// TIA Portal V19 export
FUNCTION_BLOCK "Dispenser_Main"   // FB1, LAD
TITLE = Main Block for Dispenser Element and Conveyor Running
{ S7_Optimized_Access := 'TRUE' }
// Holds Code for Dispenser Project , Light Gates and Conveyor Belt Motor.
// stored: MemoryReserve 100, SetENOAutomatically false
   VAR_TEMP   // added for the SCL form of the ladder/FBD networks
      _w1 : Bool;
   END_VAR
BEGIN

REGION Network 1: Power Up
   // Enabled Power To System
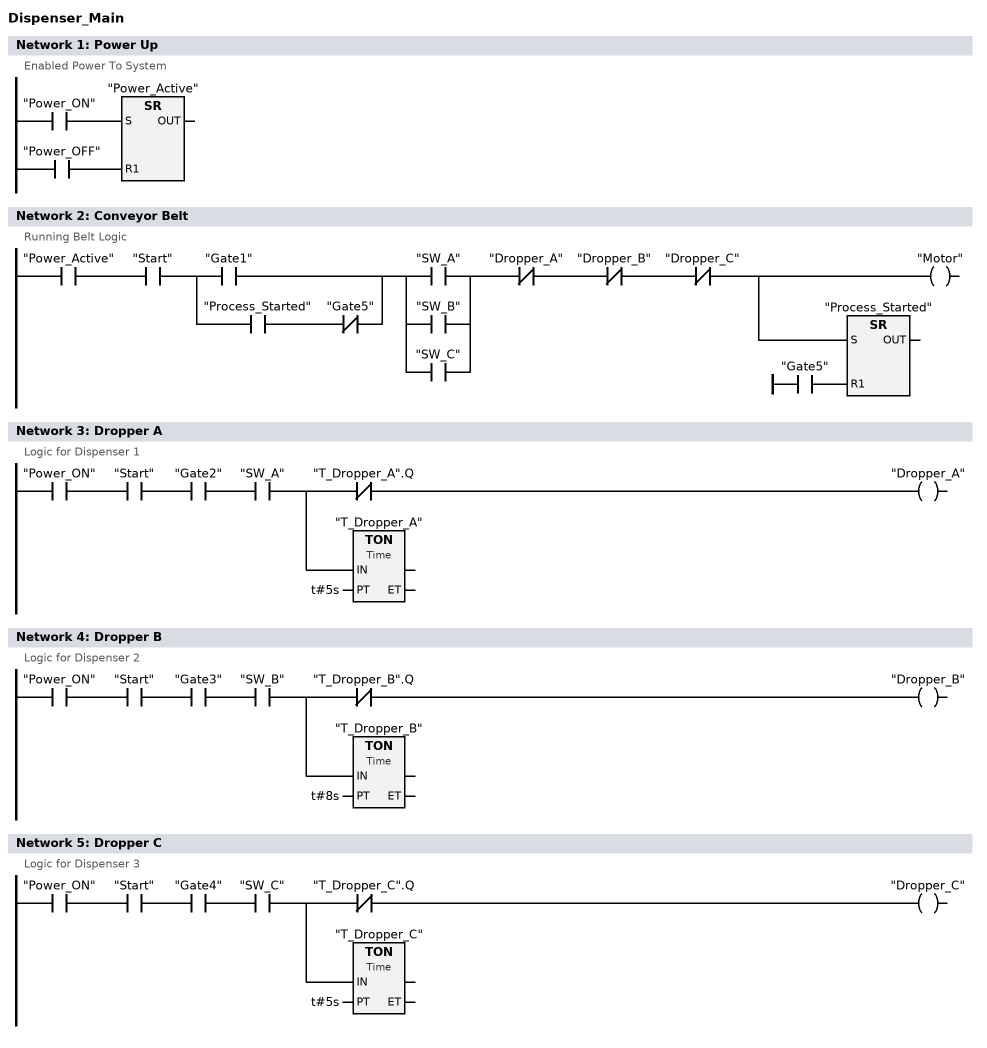
   RUNG wire#powerrail
      Contact( "Power_ON" )
      S_SR(operand := "Power_Active", r1 := wire#w1)
   END_RUNG
   RUNG wire#powerrail
      Contact( "Power_OFF" )
   END_RUNG wire#w1
   // the same network as SCL:
   IF "Power_ON" THEN
       "Power_Active" := TRUE;   // SR flip-flop
   END_IF;
   IF "Power_OFF" THEN "Power_Active" := FALSE; END_IF;
END_REGION

REGION Network 2: Conveyor Belt
   // Running Belt Logic
   RUNG wire#powerrail
      Contact( "Power_Active" )
      Contact( "Start" )
      wire#w1
      Contact( "Gate1" )
      wire#w2
      Contact( "SW_A" )
      wire#w3
      I_Contact( "Dropper_A" )
      I_Contact( "Dropper_B" )
      I_Contact( "Dropper_C" )
      wire#w4
      Coil( "Motor" )
   END_RUNG
   RUNG wire#w1
      Contact( "Process_Started" )
      I_Contact( "Gate5" )
   END_RUNG wire#w2
   RUNG wire#w2
      Contact( "SW_B" )
   END_RUNG wire#w3
   RUNG wire#w2
      Contact( "SW_C" )
   END_RUNG wire#w3
   RUNG wire#w4
      S_SR(operand := "Process_Started", r1 := wire#w5)
   END_RUNG
   RUNG wire#powerrail
      Contact( "Gate5" )
   END_RUNG wire#w5
   // the same network as SCL:
   "Motor" := "Power_Active" AND "Start" AND ("Gate1" OR ("Process_Started" AND NOT "Gate5")) AND ("SW_A" OR "SW_B" OR "SW_C") AND NOT "Dropper_A" AND NOT "Dropper_B" AND NOT "Dropper_C";
   IF "Motor" THEN
       "Process_Started" := TRUE;   // SR flip-flop
   END_IF;
   IF "Gate5" THEN "Process_Started" := FALSE; END_IF;
END_REGION

REGION Network 3: Dropper A
   // Logic for Dispenser 1
   RUNG wire#powerrail
      Contact( "Power_ON" )
      Contact( "Start" )
      Contact( "Gate2" )
      Contact( "SW_A" )
      wire#w1
      I_Contact( "T_Dropper_A".Q )
      Coil( "Dropper_A" )
   END_RUNG
   RUNG wire#w1
      { S7_Templates := "time_type := Time" } "T_Dropper_A".TON(pt := t#5s, et =>)
   END_RUNG
   // the same network as SCL:
   #_w1 := "Power_ON" AND "Start" AND "Gate2" AND "SW_A";
   "Dropper_A" := #_w1 AND NOT "T_Dropper_A".Q;
   "T_Dropper_A".TON(IN := #_w1, PT := t#5s);
END_REGION

REGION Network 4: Dropper B
   // Logic for Dispenser 2
   RUNG wire#powerrail
      Contact( "Power_ON" )
      Contact( "Start" )
      Contact( "Gate3" )
      Contact( "SW_B" )
      wire#w1
      I_Contact( "T_Dropper_B".Q )
      Coil( "Dropper_B" )
   END_RUNG
   RUNG wire#w1
      { S7_Templates := "time_type := Time" } "T_Dropper_B".TON(pt := t#8s, et =>)
   END_RUNG
   // the same network as SCL:
   #_w1 := "Power_ON" AND "Start" AND "Gate3" AND "SW_B";
   "Dropper_B" := #_w1 AND NOT "T_Dropper_B".Q;
   "T_Dropper_B".TON(IN := #_w1, PT := t#8s);
END_REGION

REGION Network 5: Dropper C
   // Logic for Dispenser 3
   RUNG wire#powerrail
      Contact( "Power_ON" )
      Contact( "Start" )
      Contact( "Gate4" )
      Contact( "SW_C" )
      wire#w1
      I_Contact( "T_Dropper_C".Q )
      Coil( "Dropper_C" )
   END_RUNG
   RUNG wire#w1
      { S7_Templates := "time_type := Time" } "T_Dropper_C".TON(pt := t#5s, et =>)
   END_RUNG
   // the same network as SCL:
   #_w1 := "Power_ON" AND "Start" AND "Gate4" AND "SW_C";
   "Dropper_C" := #_w1 AND NOT "T_Dropper_C".Q;
   "T_Dropper_C".TON(IN := #_w1, PT := t#5s);
END_REGION

REGION Network 6: Spare Network
END_REGION
END_FUNCTION_BLOCK
